FUNCTION_BLOCK DigitalOutput IMPLEMENTS I_DigitalOutput
VAR_INPUT
END_VAR
VAR_OUTPUT
END_VAR
VAR
	ID:				STRING(25);
	Output			AT%I*: BOOL;
END_VAR

METHOD FB_init : BOOL
VAR_INPUT
	bInitRetains : BOOL; // if TRUE, the retain variables are initialized (warm start / cold start)
	bInCopyCode : BOOL;  // if TRUE, the instance afterwards gets moved into the copy code (online change)
	ID:			String(25);
END_VAR
this^.ID:= ID;
END_METHOD

PROPERTY PUBLIC P_ID : String(25)
GET
P_ID:= ID;
END_GET
END_PROPERTY

PROPERTY PUBLIC P_MappingStatus : EPlcMappingStatus
GET
P_MappingStatus:= F_GetMappingStatus(ADR(Input), SIZEOF(BOOL));
END_GET
END_PROPERTY

PROPERTY PUBLIC P_Value : bool
SET // PUBLIC
Output:= P_Value;
END_SET
END_PROPERTY

END_FUNCTION_BLOCK

(* stored: Version 1.1.0.1
   POU DigitalOutput: Id {9c6c856c-bfc6-09b8-0205-5829241d18e2}, SpecialFunc None
   Method FB_init: Id {75162285-a628-0e00-3fd4-7fd09070c77b}
   Property P_ID: Id {f50a731d-33e5-019b-0fc3-26d5f1374f48}
   Get Get: Id {cfa231bf-ff32-0ded-1b81-f9ced6eebfc5}
   Property P_MappingStatus: Id {68d80066-640f-0c5e-2569-3ac4e0538722}
   Get Get: Id {9cacf2b0-ba9f-08d3-0509-bfa18adbaac4}
   Property P_Value: Id {696506a3-db60-0746-2f1d-1c14b42d34db}
   Set Set: Id {69af308d-96e0-0ca6-0d1c-c75ab3a009fc} *)
